// TIA Portal V18 export
// export: Created 2026-04-18T00:00:00Z, ExportSetting WithDefaults
FUNCTION "FC_PLC2_Logic" : Void   // FC10, LAD
{ S7_Optimized_Access := 'TRUE' }
VERSION : 0.1
// stored: AutoNumber true, IsIECCheckEnabled false
BEGIN

REGION Network 1: Freq Scale: SP x 10
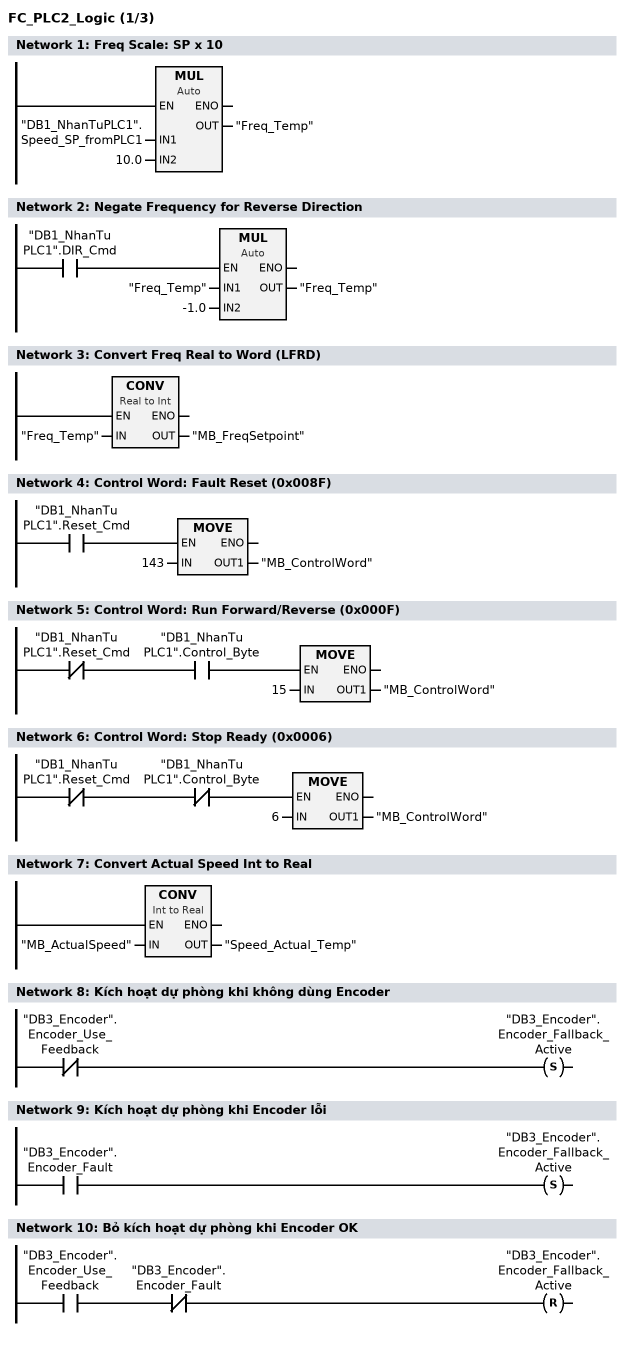
   RUNG wire#powerrail
      { S7_GenerateENO := "TRUE" } Mul(in1 := "DB1_NhanTuPLC1".Speed_SP_fromPLC1, in2 := 10.0, out => "Freq_Temp")
   END_RUNG
   // the same network as SCL:
   "Freq_Temp" := "DB1_NhanTuPLC1".Speed_SP_fromPLC1 * 10.0;
END_REGION

REGION Network 2: Negate Frequency for Reverse Direction
   RUNG wire#powerrail
      Contact( "DB1_NhanTuPLC1".DIR_Cmd )
      { S7_GenerateENO := "TRUE" } Mul(in1 := "Freq_Temp", in2 := -1.0, out => "Freq_Temp")
   END_RUNG
   // the same network as SCL:
   IF "DB1_NhanTuPLC1".DIR_Cmd THEN "Freq_Temp" := "Freq_Temp" * (-1.0); END_IF;
END_REGION

REGION Network 3: Convert Freq Real to Word (LFRD)
   RUNG wire#powerrail
      { S7_Templates := "[SrcType := Real, DestType := Int]"; S7_GenerateENO := "TRUE" } Convert(in := "Freq_Temp", out => "MB_FreqSetpoint")
   END_RUNG
   // the same network as SCL:
   "MB_FreqSetpoint" := REAL_TO_INT("Freq_Temp");
END_REGION

REGION Network 4: Control Word: Fault Reset (0x008F)
   RUNG wire#powerrail
      Contact( "DB1_NhanTuPLC1".Reset_Cmd )
      { S7_GenerateENO := "TRUE" } Move(in := 143, out1 => "MB_ControlWord")
   END_RUNG
   // the same network as SCL:
   IF "DB1_NhanTuPLC1".Reset_Cmd THEN "MB_ControlWord" := 143; END_IF;
END_REGION

REGION Network 5: Control Word: Run Forward/Reverse (0x000F)
   RUNG wire#powerrail
      I_Contact( "DB1_NhanTuPLC1".Reset_Cmd )
      Contact( "DB1_NhanTuPLC1".Control_Byte )
      { S7_GenerateENO := "TRUE" } Move(in := 15, out1 => "MB_ControlWord")
   END_RUNG
   // the same network as SCL:
   IF NOT "DB1_NhanTuPLC1".Reset_Cmd AND "DB1_NhanTuPLC1".Control_Byte THEN "MB_ControlWord" := 15; END_IF;
END_REGION

REGION Network 6: Control Word: Stop Ready (0x0006)
   RUNG wire#powerrail
      I_Contact( "DB1_NhanTuPLC1".Reset_Cmd )
      I_Contact( "DB1_NhanTuPLC1".Control_Byte )
      { S7_GenerateENO := "TRUE" } Move(in := 6, out1 => "MB_ControlWord")
   END_RUNG
   // the same network as SCL:
   IF NOT "DB1_NhanTuPLC1".Reset_Cmd AND NOT "DB1_NhanTuPLC1".Control_Byte THEN
       "MB_ControlWord" := 6;
   END_IF;
END_REGION

REGION Network 7: Convert Actual Speed Int to Real
   RUNG wire#powerrail
      { S7_Templates := "[SrcType := Int, DestType := Real]"; S7_GenerateENO := "TRUE" } Convert(in := "MB_ActualSpeed", out => "Speed_Actual_Temp")
   END_RUNG
   // the same network as SCL:
   "Speed_Actual_Temp" := INT_TO_REAL("MB_ActualSpeed");
END_REGION

REGION Network 8: Kích hoạt dự phòng khi không dùng Encoder
   RUNG wire#powerrail
      I_Contact( "DB3_Encoder".Encoder_Use_Feedback )
      S_Coil( "DB3_Encoder".Encoder_Fallback_Active )
   END_RUNG
   // the same network as SCL:
   IF NOT "DB3_Encoder".Encoder_Use_Feedback THEN "DB3_Encoder".Encoder_Fallback_Active := TRUE; END_IF;
END_REGION

REGION Network 9: Kích hoạt dự phòng khi Encoder lỗi
   RUNG wire#powerrail
      Contact( "DB3_Encoder".Encoder_Fault )
      S_Coil( "DB3_Encoder".Encoder_Fallback_Active )
   END_RUNG
   // the same network as SCL:
   IF "DB3_Encoder".Encoder_Fault THEN "DB3_Encoder".Encoder_Fallback_Active := TRUE; END_IF;
END_REGION

REGION Network 10: Bỏ kích hoạt dự phòng khi Encoder OK
   RUNG wire#powerrail
      Contact( "DB3_Encoder".Encoder_Use_Feedback )
      I_Contact( "DB3_Encoder".Encoder_Fault )
      R_Coil( "DB3_Encoder".Encoder_Fallback_Active )
   END_RUNG
   // the same network as SCL:
   IF "DB3_Encoder".Encoder_Use_Feedback AND NOT "DB3_Encoder".Encoder_Fault THEN
       "DB3_Encoder".Encoder_Fallback_Active := FALSE;
   END_IF;
END_REGION

REGION Network 11: Gửi tốc độ thực về PLC_1 chế độ bình thường
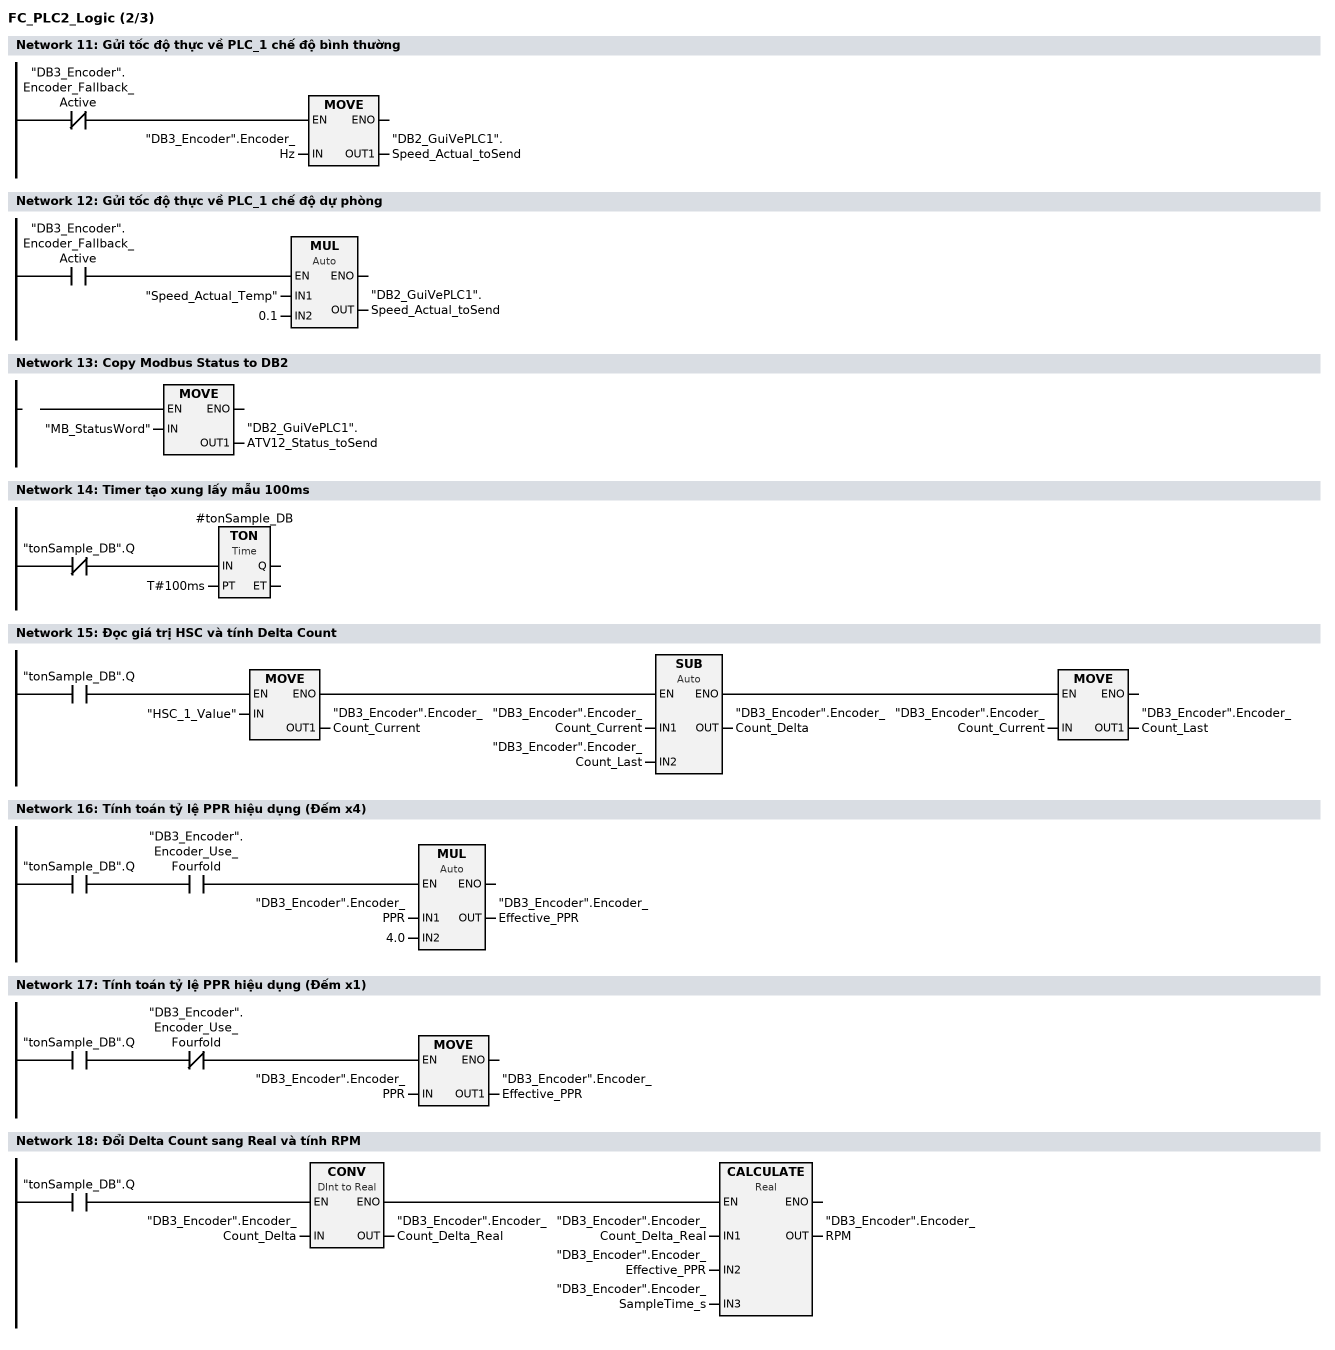
   RUNG wire#powerrail
      I_Contact( "DB3_Encoder".Encoder_Fallback_Active )
      { S7_GenerateENO := "TRUE" } Move(in := "DB3_Encoder".Encoder_Hz, out1 => "DB2_GuiVePLC1".Speed_Actual_toSend)
   END_RUNG
   // the same network as SCL:
   IF NOT "DB3_Encoder".Encoder_Fallback_Active THEN
       "DB2_GuiVePLC1".Speed_Actual_toSend := "DB3_Encoder".Encoder_Hz;
   END_IF;
END_REGION

REGION Network 12: Gửi tốc độ thực về PLC_1 chế độ dự phòng
   RUNG wire#powerrail
      Contact( "DB3_Encoder".Encoder_Fallback_Active )
      { S7_GenerateENO := "TRUE" } Mul(in1 := "Speed_Actual_Temp", in2 := 0.1, out => "DB2_GuiVePLC1".Speed_Actual_toSend)
   END_RUNG
   // the same network as SCL:
   IF "DB3_Encoder".Encoder_Fallback_Active THEN
       "DB2_GuiVePLC1".Speed_Actual_toSend := "Speed_Actual_Temp" * 0.1;
   END_IF;
END_REGION

REGION Network 13: Copy Modbus Status to DB2
   // no checked SCL form for this network; see the picture
END_REGION

REGION Network 14: Timer tạo xung lấy mẫu 100ms
   RUNG wire#powerrail
      I_Contact( "tonSample_DB".Q )
      { S7_Templates := "time_type := Time" } #tonSample_DB.TON(pt := T#100ms, et =>)
   END_RUNG
   // the same network as SCL:
   #tonSample_DB.TON(IN := NOT "tonSample_DB".Q, PT := T#100ms);
END_REGION

REGION Network 15: Đọc giá trị HSC và tính Delta Count
   RUNG wire#powerrail
      Contact( "tonSample_DB".Q )
      { S7_GenerateENO := "TRUE" } Move(in := "HSC_1_Value", out1 => "DB3_Encoder".Encoder_Count_Current)
      { S7_GenerateENO := "TRUE" } Sub(in1 := "DB3_Encoder".Encoder_Count_Current, in2 := "DB3_Encoder".Encoder_Count_Last, out => "DB3_Encoder".Encoder_Count_Delta)
      { S7_GenerateENO := "TRUE" } Move(in := "DB3_Encoder".Encoder_Count_Current, out1 => "DB3_Encoder".Encoder_Count_Last)
   END_RUNG
   // the same network as SCL:
   // ENO of a box is taken as its EN; it also drops when the box reports an error
   IF "tonSample_DB".Q THEN
       "DB3_Encoder".Encoder_Count_Current := "HSC_1_Value";
       "DB3_Encoder".Encoder_Count_Delta := "DB3_Encoder".Encoder_Count_Current - "DB3_Encoder".Encoder_Count_Last;
       "DB3_Encoder".Encoder_Count_Last := "DB3_Encoder".Encoder_Count_Current;
   END_IF;
END_REGION

REGION Network 16: Tính toán tỷ lệ PPR hiệu dụng (Đếm x4)
   RUNG wire#powerrail
      Contact( "tonSample_DB".Q )
      Contact( "DB3_Encoder".Encoder_Use_Fourfold )
      { S7_GenerateENO := "TRUE" } Mul(in1 := "DB3_Encoder".Encoder_PPR, in2 := 4.0, out => "DB3_Encoder".Encoder_Effective_PPR)
   END_RUNG
   // the same network as SCL:
   IF "tonSample_DB".Q AND "DB3_Encoder".Encoder_Use_Fourfold THEN
       "DB3_Encoder".Encoder_Effective_PPR := "DB3_Encoder".Encoder_PPR * 4.0;
   END_IF;
END_REGION

REGION Network 17: Tính toán tỷ lệ PPR hiệu dụng (Đếm x1)
   RUNG wire#powerrail
      Contact( "tonSample_DB".Q )
      I_Contact( "DB3_Encoder".Encoder_Use_Fourfold )
      { S7_GenerateENO := "TRUE" } Move(in := "DB3_Encoder".Encoder_PPR, out1 => "DB3_Encoder".Encoder_Effective_PPR)
   END_RUNG
   // the same network as SCL:
   IF "tonSample_DB".Q AND NOT "DB3_Encoder".Encoder_Use_Fourfold THEN
       "DB3_Encoder".Encoder_Effective_PPR := "DB3_Encoder".Encoder_PPR;
   END_IF;
END_REGION

REGION Network 18: Đổi Delta Count sang Real và tính RPM
   RUNG wire#powerrail
      Contact( "tonSample_DB".Q )
      { S7_Templates := "[SrcType := DInt, DestType := Real]"; S7_GenerateENO := "TRUE" } Convert(in := "DB3_Encoder".Encoder_Count_Delta, out => "DB3_Encoder".Encoder_Count_Delta_Real)
      { S7_Templates := "SrcType := Real"; S7_GenerateENO := "TRUE"; S7_Expression := "(IN1 * 60.0) / (IN2 * IN3)" } Calculate(in1 := "DB3_Encoder".Encoder_Count_Delta_Real, in2 := "DB3_Encoder".Encoder_Effective_PPR, in3 := "DB3_Encoder".Encoder_SampleTime_s, out => "DB3_Encoder".Encoder_RPM)
   END_RUNG
   // the same network as SCL:
   // ENO of a box is taken as its EN; it also drops when the box reports an error
   IF "tonSample_DB".Q THEN
       "DB3_Encoder".Encoder_Count_Delta_Real := DINT_TO_REAL("DB3_Encoder".Encoder_Count_Delta);
       "DB3_Encoder".Encoder_RPM := ("DB3_Encoder".Encoder_Count_Delta_Real * 60.0) / ("DB3_Encoder".Encoder_Effective_PPR * "DB3_Encoder".Encoder_SampleTime_s);
   END_IF;
END_REGION

REGION Network 19: Tính tần số Hz và lọc thông thấp
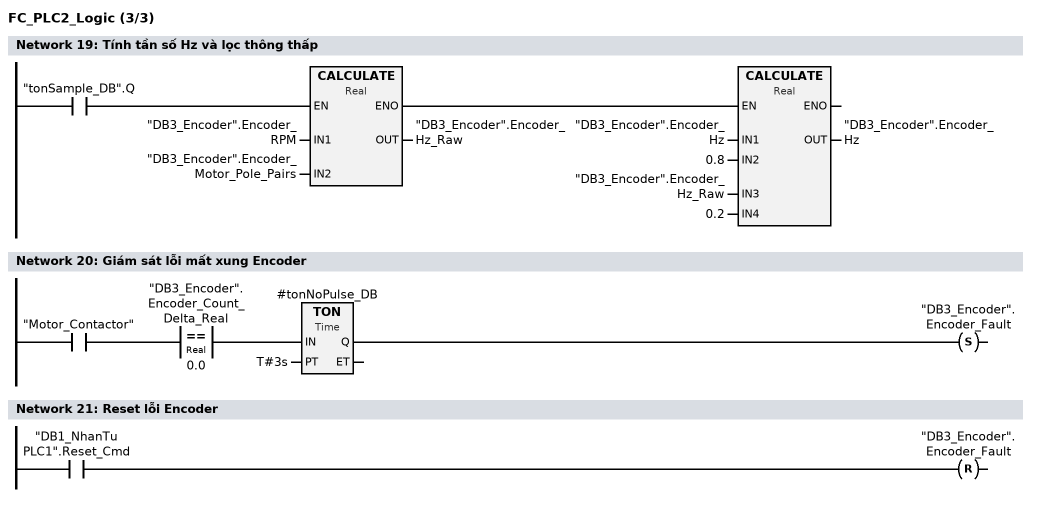
   RUNG wire#powerrail
      Contact( "tonSample_DB".Q )
      { S7_Templates := "SrcType := Real"; S7_GenerateENO := "TRUE"; S7_Expression := "(IN1 * IN2) / 60.0" } Calculate(in1 := "DB3_Encoder".Encoder_RPM, in2 := "DB3_Encoder".Encoder_Motor_Pole_Pairs, out => "DB3_Encoder".Encoder_Hz_Raw)
      { S7_Templates := "SrcType := Real"; S7_GenerateENO := "TRUE"; S7_Expression := "IN1*IN2 + IN3*IN4" } Calculate(in1 := "DB3_Encoder".Encoder_Hz, in2 := 0.8, in3 := "DB3_Encoder".Encoder_Hz_Raw, in4 := 0.2, out => "DB3_Encoder".Encoder_Hz)
   END_RUNG
   // the same network as SCL:
   // ENO of a box is taken as its EN; it also drops when the box reports an error
   IF "tonSample_DB".Q THEN
       "DB3_Encoder".Encoder_Hz_Raw := ("DB3_Encoder".Encoder_RPM * "DB3_Encoder".Encoder_Motor_Pole_Pairs) / 60.0;
       "DB3_Encoder".Encoder_Hz := "DB3_Encoder".Encoder_Hz*0.8 + "DB3_Encoder".Encoder_Hz_Raw*0.2;
   END_IF;
END_REGION

REGION Network 20: Giám sát lỗi mất xung Encoder
   RUNG wire#powerrail
      Contact( "Motor_Contactor" )
      { S7_Templates := "SrcType := Real" } EQ_Contact(in1 := "DB3_Encoder".Encoder_Count_Delta_Real, in2 := 0.0)
      { S7_Templates := "time_type := Time" } #tonNoPulse_DB.TON(pt := T#3s, et =>)
      S_Coil( "DB3_Encoder".Encoder_Fault )
   END_RUNG
   // the same network as SCL:
   #tonNoPulse_DB.TON(IN := "Motor_Contactor" AND ("DB3_Encoder".Encoder_Count_Delta_Real = 0.0), PT := T#3s);
   IF #tonNoPulse_DB.Q THEN "DB3_Encoder".Encoder_Fault := TRUE; END_IF;
END_REGION

REGION Network 21: Reset lỗi Encoder
   RUNG wire#powerrail
      Contact( "DB1_NhanTuPLC1".Reset_Cmd )
      R_Coil( "DB3_Encoder".Encoder_Fault )
   END_RUNG
   // the same network as SCL:
   IF "DB1_NhanTuPLC1".Reset_Cmd THEN "DB3_Encoder".Encoder_Fault := FALSE; END_IF;
END_REGION
END_FUNCTION
